DATA_BLOCK "MES_CHeck_DB"
{ S7_Optimized_Access := 'TRUE' }
VERSION : 0.1
NON_RETAIN
// ATTRIBUTES
// AUTO_NUMBER = False
// BLOCK_NUMBER = 111
// END_ATTRIBUTES
"MES_CHeck"

BEGIN

END_DATA_BLOCK

